{attribute 'qualified_only'}
{attribute 'to_string'}
TYPE E_GCSpinAxisJogErrorCode :
(
	None := 0,
	Axis_Not_Servo_On_During_Starting,
	Axis_Is_Busy_During_Starting,
	Invalid_Param,
	Jog_Error_During_Execute,
	// The BaseUnit was already owned by another Service.
	Resource_Acquire_Failed_During_Starting
)UDINT;
END_TYPE

(* stored: Version 1.1.0.1, ProductVersion 3.1.4026.18
   DUT E_GCSpinAxisJogErrorCode: Id {d968d262-344c-4767-a699-20264793c7d1} *)
